TYPE ST_EL1918_B :
STRUCT
	//--------------------------------------------------------------------------------------------------------
	sTerminalName                  :   STRING(200):= 'EL1918 | 8-Channel Safety Digital Input';
    //============================================================================================================================	
	// TERMINAL - EL1918 8-Channel Digital Input Terminal 	(Term 5)

	iEL1918_Ch1                		AT %I*			: 	BOOL;	// EL1918 channel 1
	iEL1918_Ch2                   	AT %I*			: 	BOOL;	// EL1918 channel 2
	iEL1918_Ch3        				AT %I*	 		: 	BOOL;	// EL1918 channel 3
	iEL1918_Ch4   					AT %I*	 		: 	BOOL;	// EL1918 channel 4
	iEL1918_Ch5         			AT %I*	 		: 	BOOL;	// EL1918 channel 5 		     			
	iEL1918_Ch6 					AT %I*			: 	BOOL;	// EL1918 channel 6
	iEL1918_Ch7               		AT %I*          :   BOOL;   // EL1918 channel 7 
    iEL1918_Ch8          			AT %I*          :   BOOL;   // EL1918 channel 8
 		
	stTerminalInfo											: 	ST_Terminal_Info;

END_STRUCT
END_TYPE

(* stored: Version 1.1.0.1
   DUT ST_EL1918_B: Id {4bd7cc3f-0aa6-498b-8f10-fd98afa697ac} *)
